// --- HELPER FUNCTION: Convert seconds (Real) to HHH:MM:SS string ---
FUNCTION "FC_SecondsToTimeString" : String[9]
{ S7_Optimized_Access := 'TRUE' }
VERSION : 0.1
	VAR_INPUT
		seconds : Real;
	END_VAR
	VAR_TEMP
		totalSec : DInt;
		hours : Int;
		minutes : Int;
		secs : Int;
		h1, h2, h3, m1, m2, s1, s2 : USInt;
	END_VAR
BEGIN
	// Convert to integer seconds
	totalSec := REAL_TO_DINT(seconds);

	// Calculate hours, minutes, seconds
	hours := DINT_TO_INT(totalSec / 3600);
	minutes := DINT_TO_INT((totalSec MOD 3600) / 60);
	secs := DINT_TO_INT(totalSec MOD 60);

	// Limit to 999:59:59 max display (over 41 days)
	IF hours > 999 THEN
		hours := 999;
		minutes := 59;
		secs := 59;
	END_IF;

	// Convert to ASCII digit values (digit type USInt, like in existing code)
	h1 := UINT_TO_USINT(hours / 100);
	h2 := UINT_TO_USINT((hours MOD 100) / 10);
	h3 := UINT_TO_USINT(hours MOD 10);
	m1 := UINT_TO_USINT(minutes / 10);
	m2 := UINT_TO_USINT(minutes MOD 10);
	s1 := UINT_TO_USINT(secs / 10);
	s2 := UINT_TO_USINT(secs MOD 10);

	// Build string "HHH:MM:SS" using BYTE_TO_CHAR like existing filename code
	#FC_SecondsToTimeString := CONCAT(IN1 := BYTE_TO_CHAR(48 + h1), IN2 := BYTE_TO_CHAR(48 + h2));
	#FC_SecondsToTimeString := CONCAT(IN1 := #FC_SecondsToTimeString, IN2 := BYTE_TO_CHAR(48 + h3));
	#FC_SecondsToTimeString := CONCAT(IN1 := #FC_SecondsToTimeString, IN2 := ':');
	#FC_SecondsToTimeString := CONCAT(IN1 := #FC_SecondsToTimeString, IN2 := BYTE_TO_CHAR(48 + m1));
	#FC_SecondsToTimeString := CONCAT(IN1 := #FC_SecondsToTimeString, IN2 := BYTE_TO_CHAR(48 + m2));
	#FC_SecondsToTimeString := CONCAT(IN1 := #FC_SecondsToTimeString, IN2 := ':');
	#FC_SecondsToTimeString := CONCAT(IN1 := #FC_SecondsToTimeString, IN2 := BYTE_TO_CHAR(48 + s1));
	#FC_SecondsToTimeString := CONCAT(IN1 := #FC_SecondsToTimeString, IN2 := BYTE_TO_CHAR(48 + s2));
END_FUNCTION

// --- LOGGING FUNCTION BLOCK ---
// Volani:
//   OB30 (1000ms): LogManager.SampleStep()   - plni buffer kazdych SampleEveryN_Cycles cyklu
//   Main (OB1):   LogManager.FlushPending   - zkontroluj flag a zapis na SD
FUNCTION_BLOCK "FB_LogManager"
{ S7_Optimized_Access := 'TRUE' }
VERSION : 0.1
	VAR_INPUT
		Enable : Bool;                     // povoleni logovani (z DB_LogConfig.Enable)
		StartTest : Bool;                  // hrana = start testu (z DB_LogConfig.StartTest)
		StopTest : Bool;                   // hrana = manual stop testu (z DB_LogConfig.StopTest)
		RPM : Real;                        // aktualni otacky vretene [RPM]
		T_Lozisko : Real;                  // teplota loziska [degC]
		T_Uhliky : Real;                   // teplota uhliku/kartacu [degC] – zatim 0.0
		Vibrace : Real;                    // vibrace – zatim 0.0
		ProudUhliky : Real;                // proud do uhliku [A], prepocitany z AQ1_CurrentCtrl_V
		State : USInt;                     // stav vretene: 0=STOP 1=RUN 2=STOPPING 3=TRIP
		RunLatched : Bool;                 // vreteno v provozu (latch z FB_DriveCtrl)
		TripActive : Bool;                 // safety trip aktivni
		TripCode : USInt;                  // kod tripu: 0=OK 1=ESTOP 2=RELAY 3=EXT 4=TEMP 5=VIB 6=DISABLE
		SafetyText : String[40];           // textova diagnostika safety brany
		SampleEveryN_Cycles : Int := 6;    // pocet cyklu OB30 mezi vzorky → 6×1s = 6s/vzorek
		TestDuration_s : DInt := 1814400;  // max delka testu [s] – timeout vypnut, beha do manualniko stopu
		FlushEveryN : Int := 5;            // pocet vzorku pred flushem: 5=test (30s), 100=produkce (10min)
		AckFlush : Bool;                   // potvrzeni flushe od FB_LogFlushToSd → resetuje FlushPending
	END_VAR

	VAR_OUTPUT
		FlushPending : Bool;       // TRUE = buffer ma dost dat → OB1 ma zapsat na SD
		TestTimeoutReached : Bool; // TRUE = test dosahl TestDuration_s (logika vypnuta)
		CyclesProcessed : DInt;    // pocet OB30 cyklu zpracovanych behem testu
		LastFlushTrigger : USInt;  // co spustilo posledni flush: 1=periodic 2=manual stop 3=timeout
		EdgeStopDetected : Bool;   // prave detekovan StopTest puls (jeden OB30 cyklus)
		EdgeStartDetected : Bool;  // prave detekovan StartTest puls (jeden OB30 cyklus)
	END_VAR

	VAR
		prevStartTest : Bool := FALSE;
		prevStopTest : Bool := FALSE;
		cycleCounter : Int := 0;
		flushCounter : Int := 0;
		StopReason : USInt := 0;  // 0=running, 1=manual stop, 2=timeout, 3=trip/fault
	END_VAR

	VAR_TEMP
		startDtl  : DTL;
		rdRet     : Int;
		yr2       : UInt;
		fName     : String[32];
		digit     : USInt;
	END_VAR

BEGIN
	// Detekce startu testu (hrana)
	EdgeStartDetected := FALSE;
	EdgeStopDetected := FALSE;

	IF Enable AND (StartTest AND NOT prevStartTest) THEN
		EdgeStartDetected := TRUE;  // Diagnostika
		"DB_LogRuntime".TestActive := TRUE;
		"DB_LogRuntime".StopSequenceActive := FALSE;
		"DB_LogRuntime".LastStopLogSaved := FALSE;
		"DB_LogRuntime".Elapsed_s := 0.0;
		"DB_LogRuntime".SampleCounter := 0;
		"DB_LogRuntime".FlushErrorCount := 0;
		"DB_LogRuntime".LastFlushOk := FALSE;  // Jeste neprobehl zadny flush
		"DB_LogRuntime".HeaderWritten := FALSE;
		"DB_LogBuffer".TrendWriteIdx := 0;
		"DB_LogBuffer".TrendReadIdx := 0;
		cycleCounter := 0;
		flushCounter := 0;
		FlushPending := FALSE;
		TestTimeoutReached := FALSE;
		CyclesProcessed := 0;  // Reset diagnostiky
		LastFlushTrigger := 0;

		// Format initial times for HMI display
		"DB_LogRuntime".ElapsedTime_HMI := '000:00:00';
		"DB_LogRuntime".TargetTime_HMI := "FC_SecondsToTimeString"(seconds := DINT_TO_REAL(TestDuration_s));

		// Generate timestamp-based file name using direct digit manipulation
		rdRet := RD_SYS_T(OUT := startDtl);

		// Build filename: LOG_YYMMDD_HHMMSS.csv
		fName := 'LOG_';

		// Year (last 2 digits)
		yr2 := startDtl.YEAR MOD 100;
		digit := UINT_TO_USINT(yr2 / 10);
		fName := CONCAT(IN1 := fName, IN2 := BYTE_TO_CHAR(48 + digit));
		digit := UINT_TO_USINT(yr2 MOD 10);
		fName := CONCAT(IN1 := fName, IN2 := BYTE_TO_CHAR(48 + digit));

		// Month
		digit := startDtl.MONTH / 10;
		fName := CONCAT(IN1 := fName, IN2 := BYTE_TO_CHAR(48 + digit));
		digit := startDtl.MONTH MOD 10;
		fName := CONCAT(IN1 := fName, IN2 := BYTE_TO_CHAR(48 + digit));

		// Day
		digit := startDtl.DAY / 10;
		fName := CONCAT(IN1 := fName, IN2 := BYTE_TO_CHAR(48 + digit));
		digit := startDtl.DAY MOD 10;
		fName := CONCAT(IN1 := fName, IN2 := BYTE_TO_CHAR(48 + digit));

		fName := CONCAT(IN1 := fName, IN2 := '_');

		// Hour
		digit := startDtl.HOUR / 10;
		fName := CONCAT(IN1 := fName, IN2 := BYTE_TO_CHAR(48 + digit));
		digit := startDtl.HOUR MOD 10;
		fName := CONCAT(IN1 := fName, IN2 := BYTE_TO_CHAR(48 + digit));

		// Minute
		digit := startDtl.MINUTE / 10;
		fName := CONCAT(IN1 := fName, IN2 := BYTE_TO_CHAR(48 + digit));
		digit := startDtl.MINUTE MOD 10;
		fName := CONCAT(IN1 := fName, IN2 := BYTE_TO_CHAR(48 + digit));

		// Second
		digit := startDtl.SECOND / 10;
		fName := CONCAT(IN1 := fName, IN2 := BYTE_TO_CHAR(48 + digit));
		digit := startDtl.SECOND MOD 10;
		fName := CONCAT(IN1 := fName, IN2 := BYTE_TO_CHAR(48 + digit));

		fName := CONCAT(IN1 := fName, IN2 := '.csv');

		"DB_LogRuntime".FileName := fName;
		"DB_LogRuntime".HeaderWritten := FALSE;
		"DB_LogRuntime".FlushErrorCount := 0;
		"DB_LogRuntime".LastFlushOk := FALSE;  // Jeste neprobehl zadny flush
		"DB_LogRuntime".MaxTempLozisko_C := 0.0;  // Reset max teploty pri startu testu
		"DB_LogRuntime".MaxTempUhliky_C := 0.0;   // Reset max teploty pri startu testu
		StopReason := 0;  // Reset stop reason - test běží
		// (event log: TEST_START)
	END_IF;

	// Detekce stopu testu (hrana)
	IF Enable AND (StopTest AND NOT prevStopTest) THEN
		EdgeStopDetected := TRUE;  // Diagnostika
		"DB_LogRuntime".StopSequenceActive := TRUE;
		"DB_LogRuntime".LastStopLogSaved := FALSE;
		StopReason := 1;  // Manual stop

		// Write final stop record before clearing TestActive so CSV captures stop state
		"DB_LogBuffer".TrendBuffer["DB_LogBuffer".TrendWriteIdx].t_s := "DB_LogRuntime".Elapsed_s;
		"DB_LogBuffer".TrendBuffer["DB_LogBuffer".TrendWriteIdx].RPM := RPM;
		"DB_LogBuffer".TrendBuffer["DB_LogBuffer".TrendWriteIdx].T_Lozisko := T_Lozisko;
		"DB_LogBuffer".TrendBuffer["DB_LogBuffer".TrendWriteIdx].T_Uhliky := T_Uhliky;
		"DB_LogBuffer".TrendBuffer["DB_LogBuffer".TrendWriteIdx].Vibrace := Vibrace;
		"DB_LogBuffer".TrendBuffer["DB_LogBuffer".TrendWriteIdx].ProudUhliky := ProudUhliky;
		"DB_LogBuffer".TrendBuffer["DB_LogBuffer".TrendWriteIdx].State := State;
		"DB_LogBuffer".TrendBuffer["DB_LogBuffer".TrendWriteIdx].RunLatched := RunLatched;
		"DB_LogBuffer".TrendBuffer["DB_LogBuffer".TrendWriteIdx].TripActive := TripActive;
		"DB_LogBuffer".TrendBuffer["DB_LogBuffer".TrendWriteIdx].TripCode := TripCode;
		"DB_LogBuffer".TrendBuffer["DB_LogBuffer".TrendWriteIdx].SafetyText := SafetyText;
		"DB_LogBuffer".TrendBuffer["DB_LogBuffer".TrendWriteIdx].TestActive := FALSE;
		"DB_LogBuffer".TrendBuffer["DB_LogBuffer".TrendWriteIdx].StopReason := StopReason;
		"DB_LogBuffer".TrendWriteIdx := "DB_LogBuffer".TrendWriteIdx + 1;
		IF "DB_LogBuffer".TrendWriteIdx > 999 THEN
			"DB_LogBuffer".TrendWriteIdx := 0;
		END_IF;

		"DB_LogRuntime".TestActive := FALSE;
		FlushPending := TRUE;   // finalni flush pri manuálním stopu
		LastFlushTrigger := 2;  // manual stop flush
		// (event log: TEST_STOP)
	END_IF;

	prevStartTest := StartTest;
	prevStopTest := StopTest;

	// Handshake: FB_LogFlushToSd potvrdil flush -> resetovat FlushPending
	// AckFlush zustane TRUE dokud FlushPending neklesne (4-way handshake)
	IF AckFlush THEN
		FlushPending := FALSE;
		flushCounter := 0;  // Reset counter az PO dokonceni flush-u
	END_IF;

	// Cyklické vzorkování pouze pokud test běží
	IF Enable AND "DB_LogRuntime".TestActive THEN
		cycleCounter := cycleCounter + 1;

		// Timer HMI se aktualizuje kazdy OB30 cyklus (1 s), nezavisle na vzorkovani logu.
		"DB_LogRuntime".Elapsed_s := "DB_LogRuntime".Elapsed_s + 1.0;
		"DB_LogRuntime".ElapsedTime_HMI := "FC_SecondsToTimeString"(seconds := "DB_LogRuntime".Elapsed_s);
		"DB_LogRuntime".TimeDisplay_HMI := CONCAT(
			IN1 := "DB_LogRuntime".ElapsedTime_HMI,
			IN2 := ' / '
		);
		"DB_LogRuntime".TimeDisplay_HMI := CONCAT(
			IN1 := "DB_LogRuntime".TimeDisplay_HMI,
			IN2 := "DB_LogRuntime".TargetTime_HMI
		);

		IF cycleCounter >= SampleEveryN_Cycles THEN
			cycleCounter := 0;

			// Zapis vzorku do kruhoveho bufferu
			"DB_LogBuffer".TrendBuffer["DB_LogBuffer".TrendWriteIdx].t_s := "DB_LogRuntime".Elapsed_s;
			"DB_LogBuffer".TrendBuffer["DB_LogBuffer".TrendWriteIdx].RPM := RPM;
			"DB_LogBuffer".TrendBuffer["DB_LogBuffer".TrendWriteIdx].T_Lozisko := T_Lozisko;
			"DB_LogBuffer".TrendBuffer["DB_LogBuffer".TrendWriteIdx].T_Uhliky := T_Uhliky;
			"DB_LogBuffer".TrendBuffer["DB_LogBuffer".TrendWriteIdx].Vibrace := Vibrace;
			"DB_LogBuffer".TrendBuffer["DB_LogBuffer".TrendWriteIdx].ProudUhliky := ProudUhliky;
			"DB_LogBuffer".TrendBuffer["DB_LogBuffer".TrendWriteIdx].State := State;
			"DB_LogBuffer".TrendBuffer["DB_LogBuffer".TrendWriteIdx].RunLatched := RunLatched;
			"DB_LogBuffer".TrendBuffer["DB_LogBuffer".TrendWriteIdx].TripActive := TripActive;
			"DB_LogBuffer".TrendBuffer["DB_LogBuffer".TrendWriteIdx].TripCode := TripCode;
			"DB_LogBuffer".TrendBuffer["DB_LogBuffer".TrendWriteIdx].SafetyText := SafetyText;
			"DB_LogBuffer".TrendBuffer["DB_LogBuffer".TrendWriteIdx].TestActive := "DB_LogRuntime".TestActive;
			"DB_LogBuffer".TrendBuffer["DB_LogBuffer".TrendWriteIdx].StopReason := StopReason;

			// Update maximalni teploty behem testu
			IF T_Lozisko > "DB_LogRuntime".MaxTempLozisko_C THEN
				"DB_LogRuntime".MaxTempLozisko_C := T_Lozisko;
			END_IF;
			IF T_Uhliky > "DB_LogRuntime".MaxTempUhliky_C THEN
				"DB_LogRuntime".MaxTempUhliky_C := T_Uhliky;
			END_IF;

			// Posun indexu (kruhový buffer)
			"DB_LogBuffer".TrendWriteIdx := "DB_LogBuffer".TrendWriteIdx + 1;
			IF "DB_LogBuffer".TrendWriteIdx > 999 THEN
				"DB_LogBuffer".TrendWriteIdx := 0;
			END_IF;
			"DB_LogRuntime".SampleCounter := "DB_LogRuntime".SampleCounter + 1;

			// FlushPending: Main vi, ze je cas zapsat na SD
			flushCounter := flushCounter + 1;
			IF flushCounter >= FlushEveryN AND NOT FlushPending THEN
				FlushPending := TRUE;
				LastFlushTrigger := 1;  // periodic flush
			END_IF;
		END_IF;

		// Konec testu po uplynutí času - VYPNUTO (test bezi do nekonecna, az do manualniho stopu)
		// IF "DB_LogRuntime".Elapsed_s >= DINT_TO_REAL(TestDuration_s) THEN
		// 	"DB_LogRuntime".TestActive := FALSE;
		// 	StopReason := 2;  // Timeout
		// 	TestTimeoutReached := TRUE;
		// 	FlushPending := TRUE;   // posledni flush
		// 	LastFlushTrigger := 3;  // timeout flush
		// 	// (event log: TEST_END_TIMEOUT)
		// END_IF;

		CyclesProcessed := CyclesProcessed + 1;  // Diagnostika
	END_IF;
END_FUNCTION_BLOCK
TYPE "UDT_SENSORS"
VERSION : 0.1
   STRUCT
      AI1_Teplota_Lozisko_C : Real;
      AI2_Teplota_Kartace_C : Real;
      TM_Rotation_A_Channel : Real;
   END_STRUCT;


END_TYPE

// --- LOGGING UDTs ---
TYPE "UDT_LogRecord"
VERSION : 0.1
	STRUCT
		t_s : Real;
		RPM : Real;
		T_Lozisko : Real;
		T_Uhliky : Real;
		Vibrace : Real;
		ProudUhliky : Real;
		State : USInt;
		RunLatched : Bool;
		TripActive : Bool;
		TripCode : USInt;
		SafetyText : String[40];
		TestActive : Bool;    // TRUE = test běží, FALSE = test byl zastaven
		StopReason : USInt;   // 0=běží, 1=manual stop, 2=timeout, 3=trip/fault
	END_STRUCT;
END_TYPE

TYPE "UDT_EventRecord"
VERSION : 0.1
	STRUCT
		t_s : Real;
		EventCode : USInt;
		EventText : String[32];
		State : USInt;
		TripCode : USInt;
		SafetyText : String[40];
	END_STRUCT;
END_TYPE

FUNCTION "FC_LogRecordToCsv" : String[254]
{ S7_Optimized_Access := 'TRUE' }
VERSION : 0.1
	VAR_INPUT
		Rec : "UDT_LogRecord";
	END_VAR

	VAR_TEMP
		line : String[254];
	END_VAR

BEGIN
	line := REAL_TO_STRING(Rec.t_s);
	line := CONCAT(IN1 := line, IN2 := ',');
	line := CONCAT(IN1 := line, IN2 := REAL_TO_STRING(Rec.RPM));
	line := CONCAT(IN1 := line, IN2 := ',');
	line := CONCAT(IN1 := line, IN2 := REAL_TO_STRING(Rec.T_Lozisko));
	line := CONCAT(IN1 := line, IN2 := ',');
	line := CONCAT(IN1 := line, IN2 := REAL_TO_STRING(Rec.T_Uhliky));
	line := CONCAT(IN1 := line, IN2 := ',');
	line := CONCAT(IN1 := line, IN2 := REAL_TO_STRING(Rec.Vibrace));
	line := CONCAT(IN1 := line, IN2 := ',');
	line := CONCAT(IN1 := line, IN2 := REAL_TO_STRING(Rec.ProudUhliky));
	line := CONCAT(IN1 := line, IN2 := ',');
	line := CONCAT(IN1 := line, IN2 := USINT_TO_STRING(Rec.State));
	line := CONCAT(IN1 := line, IN2 := ',');

	IF Rec.RunLatched THEN
		line := CONCAT(IN1 := line, IN2 := '1');
	ELSE
		line := CONCAT(IN1 := line, IN2 := '0');
	END_IF;

	line := CONCAT(IN1 := line, IN2 := ',');
	IF Rec.TripActive THEN
		line := CONCAT(IN1 := line, IN2 := '1');
	ELSE
		line := CONCAT(IN1 := line, IN2 := '0');
	END_IF;

	line := CONCAT(IN1 := line, IN2 := ',');
	line := CONCAT(IN1 := line, IN2 := USINT_TO_STRING(Rec.TripCode));
	line := CONCAT(IN1 := line, IN2 := ',');
	line := CONCAT(IN1 := line, IN2 := Rec.SafetyText);
	line := CONCAT(IN1 := line, IN2 := ',');

	IF Rec.TestActive THEN
		line := CONCAT(IN1 := line, IN2 := '1');
	ELSE
		line := CONCAT(IN1 := line, IN2 := '0');
	END_IF;

	line := CONCAT(IN1 := line, IN2 := ',');
	line := CONCAT(IN1 := line, IN2 := USINT_TO_STRING(Rec.StopReason));

	#FC_LogRecordToCsv := #line;
END_FUNCTION

DATA_BLOCK "DB_LogConfig"
{ S7_Optimized_Access := 'TRUE' }
VERSION : 0.1
NON_RETAIN
	VAR
		Enable : Bool;             // TRUE = logovani povoleno (default TRUE)
		StartTest : Bool;          // HMI/WebAPI: nastav TRUE pro start testu (hrana, auto-reset OB30)
		StopTest : Bool;           // HMI/WebAPI: nastav TRUE pro manual stop testu (hrana, auto-reset OB30)
		TestDuration_s : DInt;     // max delka testu [s] – default 1814400 = 3 tydny
		FlushEveryN : Int;         // flush kazdych N vzorku – default 5 (30s), prod 100 (10min)
		FilePrefix : String[16];   // rezerva pro pojmenovani souboru (zatim nevyuzito)
	END_VAR
BEGIN
	Enable := TRUE;
	StartTest := false;
	StopTest := false;
	TestDuration_s := 1814400;  // 3 tydny = 21 dni = 504 hodin
	FlushEveryN := 5;  // TESTOVACI NASTAVENI (prod: 100)
	FilePrefix := 'testlog';
END_DATA_BLOCK

DATA_BLOCK "DB_LogRuntime"
{ S7_Optimized_Access := 'TRUE' }
VERSION : 0.2
NON_RETAIN
	VAR
		TestActive : Bool;             // TRUE = test probiha (sleduj pro zahajeni mereni)
		TestActivePrev : Bool;         // predchozi stav TestActive pro edge logiku v OB1
		StartReqLatched : Bool;        // OB1 latch StartTest pulsu (ochrana proti ztrate hrany pri OB30=1000ms)
		StopReqLatched : Bool;         // OB1 latch StopTest pulsu (ochrana proti ztrate hrany pri OB30=1000ms)
		StopSequenceActive : Bool;     // TRUE = probiha stop sekvence a ceka se na final flush
		LastStopLogSaved : Bool;       // TRUE = posledni stop dokoncil flush na SD (indikace pro HMI)
		TestStartTs : Date_And_Time;   // cas startu testu (RD_SYS_T pri StartTest hrane)
		Elapsed_s : Real;              // uplynuly cas od startu testu [s], aktualizuje se kazdou 1s
		SampleCounter : DInt;          // celkovy pocet vzorku zapsanych do bufferu od startu
		LastFlushOk : Bool;            // TRUE = posledni flush na SD probehl bez chyby
		LastError : String[40];        // text posledni chyby flushe (FileWriteC status kod)
		FileName : String[32];         // nazev aktualniho log souboru (LOG_YYMMDD_HHMMSS.csv)
		HeaderWritten : Bool;          // TRUE = CSV hlavicka uz zapsana do souboru
		FlushErrorCount : Int;         // pocet chyb flushe od posledniho startu (alarm >0)
		// HMI display strings (formatted time)
		ElapsedTime_HMI : String[9];   // HMI zobrazeni uplynuteho casu "HHH:MM:SS" (max 999h)
		TargetTime_HMI : String[9];    // HMI zobrazeni ciloveho casu "HHH:MM:SS"
		TimeDisplay_HMI : String[21];  // HMI jedno pole: "HHH:MM:SS / HHH:MM:SS"
		// Maximalni teploty behem testu
		MaxTempLozisko_C : Real;       // max teplota loziska od startu testu [degC]
		MaxTempUhliky_C : Real;        // max teplota uhliku/kartacu od startu testu [degC]
		// OB30 cycle time monitoring
		OB30_LastTs : DTL;             // posledni cas zacatku OB30 cyklu
		OB30_CycleTime_ms : Int;       // delka aktualniho OB30 cyklu [ms]
		OB30_MaxCycleTime_ms : Int;    // maximum vzorkovany cyklus [ms]
		OB30_MinCycleTime_ms : Int;    // minimum vzorkovany cyklus [ms] (init 1000)
		OB30_AverageCycleTime_ms : Real; // prumer platnych OB30 cyklu [ms]
		OB30_CycleTimeOutOfRange : Bool; // TRUE = prumer mimo 950..1050 ms pro HMI
		OB30_CycleTimeSum_ms : Real;   // pomocny soucet platnych OB30 mereni [ms]
		OB30_CycleCounter : DInt;      // pocet OB30 cyklu od startu testu (kazdych 1s by se zvysil o 1)
	END_VAR
BEGIN
	TestActive := false;
	TestActivePrev := false;
	StartReqLatched := false;
	StopReqLatched := false;
	StopSequenceActive := false;
	LastStopLogSaved := false;
	Elapsed_s := 0.0;
	SampleCounter := 0;
	LastFlushOk := false;  // Jeste neprobehl zadny flush
	LastError := '';
	FileName := '';
	HeaderWritten := false;
	FlushErrorCount := 0;
	ElapsedTime_HMI := '000:00:00';
	TargetTime_HMI := '000:00:00';
	TimeDisplay_HMI := '000:00:00 / 000:00:00';
	MaxTempLozisko_C := 0.0;
	MaxTempUhliky_C := 0.0;
	OB30_CycleTime_ms := 0;
	OB30_MaxCycleTime_ms := 0;
	OB30_MinCycleTime_ms := 1000;
	OB30_AverageCycleTime_ms := 0.0;
	OB30_CycleTimeOutOfRange := FALSE;
	OB30_CycleTimeSum_ms := 0.0;
	OB30_CycleCounter := 0;
END_DATA_BLOCK

DATA_BLOCK "DB_LogBuffer"
{ S7_Optimized_Access := 'TRUE' }
VERSION : 0.1
NON_RETAIN
	VAR
		TrendBuffer : ARRAY[0..999] OF "UDT_LogRecord";   // kruhovy buffer vzorku (1000 polozek × 6s = 100 min)
		EventBuffer : ARRAY[0..99] OF "UDT_EventRecord";  // buffer eventu (faze 3)
		TrendWriteIdx : Int;   // index zapisu (LogManager) – sleduj pro debug plneni bufferu
		TrendReadIdx : Int;    // index cteni/flushe (LogFlushToSd) – WriteIdx-ReadIdx = neprectenych radku
		EventWriteIdx : Int;   // index zapisu eventu
		EventReadIdx : Int;    // index cteni eventu
	END_VAR
BEGIN
	TrendWriteIdx := 0;
	TrendReadIdx := 0;
	EventWriteIdx := 0;
	EventReadIdx := 0;
END_DATA_BLOCK

DATA_BLOCK "DB_HMI"
{ S7_Optimized_Access := 'TRUE' }
VERSION : 0.1
NON_RETAIN
   VAR
      Sensors { S7_SetPoint := 'False'} : "UDT_SENSORS";   // AI hodnoty po prepoctu (teploty degC, RPM)
      System : Struct
         Enable : Bool;   // rezerva pro systemove povoleni
      END_STRUCT;
      Spindle : Struct
         Start : Bool;    // HMI puls start vretene (auto-reset v OB1)
         Stop : Bool;     // HMI puls stop vretene (auto-reset v OB1)
         ResetFault : Bool;  // HMI puls reset chyby meniče
         Speed_RPM : Real;   // zadane otacky vretene [RPM] – max 18000
         Enable : Bool;      // rezerva
      END_STRUCT;
      LabPSU : Struct
         Enable : Bool;            // povoleni laboratorniho zdroje (auto-set pri StartTest)
			Cycle_s : Real;           // perioda OB30 [s] – default 1.0
			Mode : USInt;             // rezim zdroje: 0=OFF 1=CONST 2=SINE_DEBUG
			BaseVoltage_V : Real;     // napeti zdroje [V] – default 2.0
			DebugAmplitude_A : Real;  // amplituda sinusoidy [A] – default 5.0
			DebugPeriod_min : Real;   // perioda sinusoidy [min] – default 1.0 min
			CurrentOffset_A : Real;   // deprecated: v SINE_DEBUG se nepouziva
			ConstCurrent_A : Real;    // proud v CONST rezimu [A] – default 10.0
			MaxCurrent_A : Real;      // maximalni povoleny proud [A] – default 38.0
			CurrentLimitExceeded : Bool;  // TRUE = zadany proud prekrocil MaxCurrent_A
			SineCycleCounter : UDInt;     // pocet dokoncenych period sinusoidy od startu
      END_STRUCT;
   END_VAR


BEGIN
	LabPSU.Enable := false;
	LabPSU.Cycle_s := 1.0;  // OB30 = 1000ms = 1s
	LabPSU.Mode := 2;  // 2 = SINE_DEBUG (sinusova modulace)
	LabPSU.BaseVoltage_V := 2.0;
	LabPSU.DebugAmplitude_A := 5.0;
	LabPSU.DebugPeriod_min := 1.0;  // 1 minuta perioda
	LabPSU.CurrentOffset_A := 5.0;
	LabPSU.ConstCurrent_A := 10.0;  // 10 A pro CONST rezim
	LabPSU.MaxCurrent_A := 38.0;
	LabPSU.CurrentLimitExceeded := false;
	LabPSU.SineCycleCounter := 0;

END_DATA_BLOCK

TYPE "UDT_TM_COUNT"
VERSION : 0.1
   STRUCT
      MeasuredValue : Real;
   END_STRUCT;

END_TYPE

TYPE "UDT_IO_AQ"
VERSION : 0.1
   STRUCT
      SpeedVoltage : Real;
      AQ2_VoltageCtrl_V : Real;
      AQ1_CurrentCtrl_V : Real;
		AQ3_OutputOff : Real;
   END_STRUCT;

END_TYPE

TYPE "UDT_IO_AI"
VERSION : 0.1
   STRUCT
      AI1_TeplotaLoziska_Ohm : Int;
      AI2_TeplotaKartace_Ohm : Int;
   END_STRUCT;

END_TYPE

TYPE "UDT_IO_DI"
VERSION : 0.1
   STRUCT
      SafetyRelayAuxOk : Bool;
      HSC_Couter : UInt;
      EmergencyStop : Bool;
      ExternalFault : Bool;
   END_STRUCT;

END_TYPE

TYPE "UDT_IO_DQ"
VERSION : 0.1
   STRUCT
      EmergencyStop : Bool;
      EmergencyStopButtonLed : Bool;
      ResetButtonLed : Bool;
      RunForwardCmd : Bool;
      FaultResetCmd : Bool;
      MultiSpeed1 : Bool;
      ExternalFault : Bool;
   END_STRUCT;

END_TYPE

FUNCTION_BLOCK "FB_SafetyGate"
{ S7_Optimized_Access := 'TRUE' }
VERSION : 0.1
   VAR_INPUT
      Enable : Bool;   // hlavní povolení systému
      EmergencyStop : Bool;   // 1 = E-Stop aktivní
      SafetyRelayAuxOk : Bool;   // 1 = safety relé OK
      ExternalFault : Bool;   // 1 = externí chyba
      TempAlarm : Bool;   // 1 = kritická teplota
      VibAlarm : Bool;   // 1 = kritické vibrace
   END_VAR

   VAR_OUTPUT
      SafetyOk : Bool;
      PermitMotion : Bool;
      TripActive : Bool;
      TripCode : USInt;
      StatusText : String[40];
   END_VAR


BEGIN
	// hardware safety stav
	#SafetyOk := #SafetyRelayAuxOk AND NOT #EmergencyStop;

	// centrální trip
	#TripActive := (NOT #SafetyOk) OR #ExternalFault OR #TempAlarm OR #VibAlarm OR (NOT #Enable);

	// povolení pohybu
	#PermitMotion := NOT #TripActive;

	// diagnostika
	IF #EmergencyStop THEN
	    #TripCode := 1;
	    #StatusText := 'E-STOP ACTIVE';
	ELSE
		IF NOT #SafetyRelayAuxOk THEN
		    #TripCode := 2;
		    #StatusText := 'SAFETY RELAY NOT OK';
		ELSE
			IF #ExternalFault THEN
			    #TripCode := 3;
			    #StatusText := 'EXTERNAL FAULT';
			ELSE
				IF #TempAlarm THEN
				    #TripCode := 4;
				    #StatusText := 'TEMP ALARM';
				ELSE
					IF #VibAlarm THEN
					    #TripCode := 5;
					    #StatusText := 'VIBRATION ALARM';
					ELSE
						IF NOT #Enable THEN
						    #TripCode := 6;
						    #StatusText := 'SYSTEM NOT ENABLED';
						ELSE
						    #TripCode := 0;
						    #StatusText := 'READY';
						END_IF;
					END_IF;
				END_IF;
			END_IF;
		END_IF;
	END_IF;
END_FUNCTION_BLOCK

FUNCTION_BLOCK "FB_LabPSU"
{ S7_Optimized_Access := 'TRUE' }
VERSION : 0.1
   VAR_INPUT
      Enable : Bool := false;   // povolenÃ­ funkce z PLC/HMI
      PermitOutput : Bool := false;   // interlock / safety gate
      Mode : USInt := 0;   // 0=OFF, 1=CONST, 2=SINE_DEBUG ÄasovÃ¡ zÃ¡kladna
      Cycle_s : Real := 0.01;   // typicky OB35 = 10 ms zdroj - zÃ¡kladnÃ­ nastavenÃ­
      BaseVoltage_V : Real := 1.0;   // AQ2
      CurrentOffset_A : Real := 0.0;   // DC offset proudu
      DebugAmplitude_A : Real := 60.0;   // amplituda sinu pro debug
      DebugPeriod_min : Real := 10.0;   // perioda sinu v minutach (default 10 min)
      ConstCurrent_A : Real := 10.0;   // rampy
      RampUp_A_per_s : Real := 50.0;
      RampDown_A_per_s : Real := 80.0;   // parametry zdroje BK1900B
	PSU_MinVoltage_V : Real := 0.8;   // minimalni napeti pro stabilni vystup zdroje
      PSU_MaxVoltage_V : Real := 16.0;   // model 1900B
      PSU_MaxCurrent_A : Real := 60.0;   // model 1900B
      RemoteMaxCtrl_V : Real := 5.0;   // analog remote 0..5 V engineering outputs
   END_VAR

   VAR_OUTPUT
      VoltageSet_V : Real := 0.0;   // poÅ¾adovanÃ© napÄ›tÃ­ zdroje
      CurrentSet_A : Real := 0.0;   // poÅ¾adovanÃ½ current limit analog outputs for PLC IO layer
      AQ2_VoltageCtrl_V : Real := 0.0;   // 0..5 V na pin 2
      AQ3_CurrentCtrl_V : Real := 0.0;   // 0..5 V na pin 3 digital output for pin 5
	AQ_OutputOff_V : Real := 5.0;   // 0.0 V = enable, 5.0 V = output off
      State : USInt := 0;   // 0 OFF, 1 CONST, 2 SINE
      StatusText : String[40] := '';
      CurrentLimitExceeded : Bool := false;   // indikator, ze uzivatel zkusil zadat vyssi proud nez limit
      SineCycleCounter : UDInt := 0;   // pocet dokoncenych period sinusovky (pro HMI)
   END_VAR

   VAR
      phase_rad : Real := 0.0;
      omega : Real := 0.0;
      targetCurrent_A : Real := 0.0;
      sineValue : Real := 0.0;
	effectiveOffset_A : Real := 0.0;
	offsetAutoAdjusted : Bool := FALSE;
	prevMode : USInt := 0;   // Pamatuje si predchozi Mode pro detekci prechodu
   END_VAR


BEGIN
	// safety / permit
	IF (NOT #Enable) OR (NOT #PermitOutput) THEN
	    #phase_rad := 0.0;
	    #VoltageSet_V := 0.0;
	    #CurrentSet_A := 0.0;
	    #AQ2_VoltageCtrl_V := 0.0;
	    #AQ3_CurrentCtrl_V := 0.0;
	    #AQ_OutputOff_V := 5.0;
	    #State := 0;
	    #StatusText := 'SAFE OFF';
	    #CurrentLimitExceeded := false;
	    #prevMode := 0;
	    RETURN;
	END_IF;

	// reset CurrentLimitExceeded flag na zacatku cyklu
	#CurrentLimitExceeded := false;

	// vystup zdroje povolen
	#AQ_OutputOff_V := 0.0;

	// zakladni napeti
	#VoltageSet_V := #BaseVoltage_V;

	// omezeni napeti
	IF #VoltageSet_V < #PSU_MinVoltage_V THEN
	    #VoltageSet_V := #PSU_MinVoltage_V;
	END_IF;
	IF #VoltageSet_V > #PSU_MaxVoltage_V THEN
	    #VoltageSet_V := #PSU_MaxVoltage_V;
	END_IF;

	CASE #Mode OF
	    0: // OFF
	        #CurrentSet_A := 0.0;
	        #VoltageSet_V := 0.0;
	        #AQ_OutputOff_V := 5.0;
	        #State := 0;
	        #StatusText := 'OFF';

	    1: // CONST
	        #targetCurrent_A := #ConstCurrent_A;

	        // detekce prekroceni limitu - pred clampingem
	        IF #targetCurrent_A > #PSU_MaxCurrent_A THEN
	            #CurrentLimitExceeded := true;
	        END_IF;

	        IF #targetCurrent_A < 0.0 THEN
	            #targetCurrent_A := 0.0;
	        END_IF;
	        IF #targetCurrent_A > #PSU_MaxCurrent_A THEN
	            #targetCurrent_A := #PSU_MaxCurrent_A;
	        END_IF;

	        // jednoducha rampa
	        IF #CurrentSet_A < #targetCurrent_A THEN
	            #CurrentSet_A := #CurrentSet_A + (#RampUp_A_per_s * #Cycle_s);
	            IF #CurrentSet_A > #targetCurrent_A THEN
	                #CurrentSet_A := #targetCurrent_A;
	            END_IF;
	        ELSE
			IF #CurrentSet_A > #targetCurrent_A THEN
			    #CurrentSet_A := #CurrentSet_A - (#RampDown_A_per_s * #Cycle_s);
			    IF #CurrentSet_A < #targetCurrent_A THEN
			        #CurrentSet_A := #targetCurrent_A;
			    END_IF;
			END_IF;
	        END_IF;

	        #State := 1;
	        #StatusText := 'CONST';

	    2: // SINE_DEBUG
	        // Pri prvnim vstupu do SINE rezimu resetovat fazi na -pi/2, aby prubeh zacinali od 0A
	        IF #prevMode <> 2 THEN
	            #phase_rad := -1.5707963;  // -pi/2 rad, zacatek prubehu od 0 A
	            #SineCycleCounter := 0;  // reset pocitadla cyklu pri vstupu do SINE rezimu
	        END_IF;

	        // Vypocet omega z periody v minutach: omega = 2*pi / (T_min * 60)
	        IF #DebugPeriod_min > 0.0 THEN
	            #omega := 6.2831853 / (#DebugPeriod_min * 60.0); // 2*pi / (T_min * 60s)
	        ELSE
	            #omega := 0.0; // ochrana proti deleni nulou
	        END_IF;
	        #offsetAutoAdjusted := FALSE;
	        IF #prevMode <> 2 THEN
	            // Prvni vypocet po vstupu do rezimu zacne presne na 0 A.
	            #phase_rad := -1.5707963 - (#omega * #Cycle_s);
	        END_IF;

	        #phase_rad := #phase_rad + (#omega * #Cycle_s);

	        // drzet fazi v rozumnem rozsahu a pocitat dokoncene periody
	        IF #phase_rad > 6.2831853 THEN
	            #phase_rad := #phase_rad - 6.2831853;
	            #SineCycleCounter := #SineCycleCounter + 1;  // dokoncena jedna perioda
	        END_IF;

	        #sineValue := SIN(#phase_rad);

	        // Cely sinus posunuty do rozsahu 0..A.
	        // DebugAmplitude_A je maximum prubehu, CurrentOffset_A se v SINE_DEBUG nepouziva.
	        #targetCurrent_A := (#DebugAmplitude_A * 0.5)
	                          + ((#DebugAmplitude_A * 0.5) * #sineValue);

	        // detekce prekroceni limitu - pred clampingem
	        IF #targetCurrent_A > #PSU_MaxCurrent_A THEN
	            #CurrentLimitExceeded := true;
	        END_IF;

	        // current limit zdroje nemuze byt zaporny
	        IF #targetCurrent_A < 0.0 THEN
	            #targetCurrent_A := 0.0;
	        END_IF;

	        IF #targetCurrent_A > #PSU_MaxCurrent_A THEN
	            #targetCurrent_A := #PSU_MaxCurrent_A;
	        END_IF;

	        // volitelne muzes i tady nechat rampu, ale pro sinus ji vetsinou nechces moc agresivni
	        #CurrentSet_A := #targetCurrent_A;

	        #State := 2;
	        #StatusText := 'SINE DEBUG 0..A';

	    ELSE
	        #CurrentSet_A := 0.0;
	        #VoltageSet_V := 0.0;
	        #AQ_OutputOff_V := 5.0;
	        #State := 0;
	        #StatusText := 'UNKNOWN->OFF';
	END_CASE;

	// prevod engineering units -> BK remote control 0..5V

	// napeti
	IF #PSU_MaxVoltage_V > 0.0 THEN
	    #AQ2_VoltageCtrl_V := (#VoltageSet_V / #PSU_MaxVoltage_V) * #RemoteMaxCtrl_V;
	ELSE
	    #AQ2_VoltageCtrl_V := 0.0;
	END_IF;

	// proud - kalibrovany prepocet na zaklade mereni
	// I [A] = 15.92 * U [V] - 6.09  ->  U [V] = (I [A] / 15.92) + 0.383
	// Dead zone: 0.383 V
	IF #CurrentSet_A > 0.0 THEN
	    #AQ3_CurrentCtrl_V := (#CurrentSet_A / 15.92) + 0.383;
	ELSE
	    #AQ3_CurrentCtrl_V := 0.0;
	END_IF;

	// clamp
	IF #AQ2_VoltageCtrl_V < 0.0 THEN
	    #AQ2_VoltageCtrl_V := 0.0;
	END_IF;
	IF #AQ2_VoltageCtrl_V > #RemoteMaxCtrl_V THEN
	    #AQ2_VoltageCtrl_V := #RemoteMaxCtrl_V;
	END_IF;

	// clamp proudoveho ridiciho signalu
	// Dead zone: pod 0.383V zdroj nereaguje
	IF #AQ3_CurrentCtrl_V < 0.0 THEN
	    #AQ3_CurrentCtrl_V := 0.0;
	END_IF;
	IF #AQ3_CurrentCtrl_V > #RemoteMaxCtrl_V THEN
	    #AQ3_CurrentCtrl_V := #RemoteMaxCtrl_V;
	END_IF;

	// Ulozit aktualni Mode pro detekci prechodu v pristim cyklu
	#prevMode := #Mode;

END_FUNCTION_BLOCK

TYPE "UDT_LABPSU_STATUS"
VERSION : 0.1
   STRUCT
      VoltageSet_V : Real;
      CurrentSet_A : Real;
      State : USInt;
      StatusText : String[40];
   END_STRUCT;

END_TYPE

TYPE "UDT_SAFETY_STATUS"
VERSION : 0.1
   STRUCT
      SafetyOk : Bool;
      PermitMotion : Bool;
      TripActive : Bool;
      TripCode : USInt;
      StatusText : String[40];
   END_STRUCT;

END_TYPE

DATA_BLOCK "DB_IO"
{ S7_Optimized_Access := 'TRUE' }
VERSION : 0.1
NON_RETAIN
   VAR
      DQ { S7_SetPoint := 'False'} : "UDT_IO_DQ";
      DI : "UDT_IO_DI";
      AI : "UDT_IO_AI";
      TM : "UDT_TM_COUNT";
      AQ : "UDT_IO_AQ";
   END_VAR


BEGIN
	AQ.AQ3_OutputOff := 5.0;

END_DATA_BLOCK

TYPE "UDT_SPINDEL_STATUS"
VERSION : 0.1
   STRUCT
      RunLatched : Bool;
      TripActive : Bool;
      State : USInt;
      StatusText : String[40];
   END_STRUCT;

END_TYPE

FUNCTION_BLOCK "FB_DriveCtrl"
{ S7_Optimized_Access := 'TRUE' }
VERSION : 0.1
   VAR_INPUT
      HMI_Start : Bool := false;   // start command (button)
      HMI_Stop : Bool := false;   // stop command (button)
      HMI_ResetFault : Bool := false;   // reset fault (button)
      HMI_Speed_RPM : Real := 0.0;   // speed setpoint in RPM Interlocks / safety
      PermitMotion : Bool := false;   // from safety gate
      EmergencyStop : Bool := false;   // E-Stop chain
      ExternalFaultIn : Bool := false;   // external fault input Parameters
      SpeedMax_RPM : Real := 18000.0;   // max RPM corresponds to 10V
      AO_MaxVolt : Real := 10.0;   // 0..10V
      RampUp_RPM_per_s : Real := 6000.0;   // ramp up rate
      RampDown_RPM_per_s : Real := 9000.0;   // ramp down rate
      ResetPulse : Time := T#300MS;   // reset pulse length
      RequireSpeedToRun : Bool := FALSE;   // if TRUE, Start only latches when setpoint > 0 Outputs to drive
   END_VAR

   VAR_OUTPUT
      DO_RunForward : Bool := false;
      DO_FaultReset : Bool := false;
      DO_MultiSpeed1 : Bool := false;
      DO_ExternalFault : Bool := false;
      AQ1_Voltage_0_10V : Real := 0.0;   // Status for HMI/diagnostics
      RunLatched : Bool := false;   // internal run request latch
      TripActive : Bool := false;   // interlock active
      State : USInt := 0;   // 0 STOPPED, 1 RUN_CMD, 2 STOPPING, 3 TRIP
      StatusText : String[40] := '';   // Edge detection
   END_VAR

   VAR
      prevStart : Bool := false;
      prevStop : Bool := false;
      prevReset : Bool := false;
      startEdge : Bool := false;
      stopEdge : Bool := false;
      resetEdge : Bool := false;   // Ramp variables
      speedCmdRPM : Real := 0.0;
      speedRampRPM : Real := 0.0;   // Reset pulse timer
      tReset {InstructionName := 'TON_TIME'; LibVersion := '1.0'; S7_SetPoint := 'False'} : TON_TIME;   // Cycle time assumption (OB1). Use OB35 for precise timing if needed.
      cycle_s { S7_SetPoint := 'True'} : Real := 0.01;   // 10 ms default
   END_VAR


BEGIN
	    // ------------------------------------------------------------
	    // Edge detection for Start/Stop/Reset
	    // ------------------------------------------------------------
	    #startEdge := #HMI_Start AND NOT #prevStart;
	    #stopEdge := #HMI_Stop AND NOT #prevStop;
	    #resetEdge := #HMI_ResetFault AND NOT #prevReset;

	    #prevStart := #HMI_Start;
	    #prevStop := #HMI_Stop;
	    #prevReset := #HMI_ResetFault;

	    // ------------------------------------------------------------
	    // Trip / interlock
	    // Trip znamena zakaz běhu vřetene, pokud není splněna bezpečnostní podmínka. Trip = okamžité odstavení zařízení.
	    // ------------------------------------------------------------
	    #TripActive := (NOT #PermitMotion) OR #EmergencyStop OR #ExternalFaultIn;

	    // External fault output to the drive (if wired this way)
	    #DO_ExternalFault := #TripActive;

	    // ------------------------------------------------------------
	    // Sanitize setpoint
	    // Sanitize = zkontrolovat a upravit vstupní hodnotu tak, aby byla bezpečná a platná.
	    // ------------------------------------------------------------
	    #speedCmdRPM := #HMI_Speed_RPM;
	    IF #speedCmdRPM < 0.0 THEN
	        #speedCmdRPM := 0.0;
	    END_IF;
	    IF #speedCmdRPM > #SpeedMax_RPM THEN
	        #speedCmdRPM := #SpeedMax_RPM;
	    END_IF;

	    // ------------------------------------------------------------
	    // Run latch logic (Stop has priority)
	    // ------------------------------------------------------------
	    IF #TripActive THEN
	        #RunLatched := FALSE;
	    ELSE
	        IF #stopEdge OR #HMI_Stop THEN
	            #RunLatched := FALSE;
	        ELSE
	            IF #startEdge THEN
	                IF (NOT #RequireSpeedToRun) OR (#speedCmdRPM > 0.0) THEN
	                    #RunLatched := TRUE;
	                END_IF;
	            END_IF;
	        END_IF;
	    END_IF;

	    // ------------------------------------------------------------
	    // Fault reset pulse (recommended only when not running)
	    // ------------------------------------------------------------
	    #tReset(IN := (#resetEdge AND NOT #TripActive AND NOT #RunLatched),
	            PT := #ResetPulse);
	    #DO_FaultReset := #tReset.Q;

	    // ------------------------------------------------------------
	    // Defaults
	    // ------------------------------------------------------------
	    #DO_MultiSpeed1 := FALSE;

	    // ------------------------------------------------------------
	    // State (for HMI readability; no drive feedback available)
	    // ------------------------------------------------------------
	    IF #TripActive THEN
	        #State := 3; // TRIP
	    ELSE
	        IF #RunLatched THEN
	            #State := 1; // RUN_CMD
	        ELSE
	            IF #speedRampRPM > 0.0 THEN
	                #State := 2; // STOPPING (ramp down)
	            ELSE
	                #State := 0; // STOPPED
	            END_IF;
	        END_IF;
	    END_IF;

	    CASE #State OF
	        0:
	            #StatusText := 'STOPPED';
	        1:
	            #StatusText := 'RUN CMD (no feedback)';
	        2:
	            #StatusText := 'STOPPING (ramp down)';
	        3:
	            #StatusText := 'TRIP (E-Stop/Interlock)';
	        ELSE
	            #StatusText := 'UNKNOWN';
	    END_CASE;

	    // ------------------------------------------------------------
	    // Drive command + speed ramp
	    // ------------------------------------------------------------
	    IF #TripActive THEN
	        #DO_RunForward := FALSE;
	        #speedRampRPM := 0.0;
	    ELSE
	        IF #RunLatched THEN
	            #DO_RunForward := TRUE;

	            // Ramp toward setpoint (up & down)
	            IF #speedRampRPM < #speedCmdRPM THEN
	                #speedRampRPM := #speedRampRPM + (#RampUp_RPM_per_s * #cycle_s);
	                IF #speedRampRPM > #speedCmdRPM THEN
	                    #speedRampRPM := #speedCmdRPM;
	                END_IF;
	            ELSE
				IF #speedRampRPM > #speedCmdRPM THEN
				    #speedRampRPM := #speedRampRPM - (#RampDown_RPM_per_s * #cycle_s);
				    IF #speedRampRPM < #speedCmdRPM THEN
				        #speedRampRPM := #speedCmdRPM;
				    END_IF;
				END_IF;
	            END_IF;

	        ELSE
	            #DO_RunForward := FALSE;

	            // Ramp down to 0
	            IF #speedRampRPM > 0.0 THEN
	                #speedRampRPM := #speedRampRPM - (#RampDown_RPM_per_s * #cycle_s);
	                IF #speedRampRPM < 0.0 THEN
	                    #speedRampRPM := 0.0;
	                END_IF;
	            END_IF;
	        END_IF;
	    END_IF;

	    // ------------------------------------------------------------
	    // RPM -> 0..10V conversion
	    // ------------------------------------------------------------
	    IF #SpeedMax_RPM > 0.0 THEN
	        #AQ1_Voltage_0_10V := (#speedRampRPM / #SpeedMax_RPM) * #AO_MaxVolt;
	    ELSE
	        #AQ1_Voltage_0_10V := 0.0;
	    END_IF;

	    // ------------------------------------------------------------
	    // Clamp AO (Clamp znamena omezit hodnotu tak, aby zůstala v daném rozsahu (min–max))
	    //  ------------------------------------------------------------
	    IF #AQ1_Voltage_0_10V < 0.0 THEN
	        #AQ1_Voltage_0_10V := 0.0;
	    END_IF;
	    IF #AQ1_Voltage_0_10V > #AO_MaxVolt THEN
	        #AQ1_Voltage_0_10V := #AO_MaxVolt;
	    END_IF;

	    // Hard safety
	    IF #TripActive THEN
	        #AQ1_Voltage_0_10V := 0.0;
	    END_IF;

END_FUNCTION_BLOCK

FUNCTION_BLOCK "FB_SafetyButtons"
{ S7_Optimized_Access := 'TRUE' }
VERSION : 0.1
   VAR_INPUT
      DI0_AuxSafetyRelay : Bool;   // AUX ze safety relé
      DI1_SafetyButton : Bool;   // signal ze safety tlačítka
   END_VAR

   VAR_OUTPUT
      DQ1_LED : Bool;   // Cervene LED svetlo na STOP tlacitku
      DQ0_LED : Bool;   // Modre LED reset svetlo
   END_VAR


BEGIN
	// Bezpečný default
	#DQ1_LED := FALSE;
	#DQ0_LED := FALSE;

	// Vyhodnocení kombinací
	IF (NOT #DI0_AuxSafetyRelay) AND (#DI1_SafetyButton) THEN
	    // DI0 = 0, DI1 = 0
	    #DQ1_LED := TRUE;
	    #DQ0_LED := FALSE;

	ELSE
		IF (NOT #DI0_AuxSafetyRelay) AND (NOT #DI1_SafetyButton) THEN
		    // DI0 = 0, DI1 = 1
		    #DQ1_LED := FALSE;
		    #DQ0_LED := TRUE;

		ELSE
			IF #DI0_AuxSafetyRelay AND (NOT #DI1_SafetyButton) THEN
			    // DI0 = 1, DI1 = 1
			    #DQ1_LED := FALSE;
			    #DQ0_LED := FALSE;

			ELSE
				// DI0 = 1, DI1_SafetyButton = true -> relay OK, button stisknuty = E-STOP fault stav
				// cervena LED sviti
				#DQ1_LED := TRUE;
				#DQ0_LED := FALSE;
			END_IF;
		END_IF;
	END_IF;
END_FUNCTION_BLOCK

DATA_BLOCK "DB_Status"
{ S7_Optimized_Access := 'TRUE' }
VERSION : 0.1
NON_RETAIN
   VAR
      Spindel { S7_SetPoint := 'False'} : "UDT_SPINDEL_STATUS";
      Safety : "UDT_SAFETY_STATUS";
      LabPSU { S7_SetPoint := 'False'} : "UDT_LABPSU_STATUS";
      // HMI helper for status panel color (Basic Panel limitation - one tag only)
	HMI_StatusColor : USInt;  // 0=READY (green), 1=RUNNING (blue), 2=RED (error/trip), 3=AMBER (running with RPM=0)
	HMI_StatusText : String[24];  // "TEST READY" / "TEST RUNNING" / "RUNNING - RPM=0" / "READY - LOG SAVED" / "ERROR - TRIP ACTIVE"
   END_VAR


BEGIN
   HMI_StatusColor := 0;
   HMI_StatusText := 'TEST READY';
END_DATA_BLOCK

DATA_BLOCK "FB_SafetyButtons_DB"
{ S7_Optimized_Access := 'TRUE' }
VERSION : 0.1
NON_RETAIN
"FB_SafetyButtons"

BEGIN

END_DATA_BLOCK

DATA_BLOCK "Spindel"
{ S7_Optimized_Access := 'TRUE' }
VERSION : 0.1
NON_RETAIN
"FB_DriveCtrl"

BEGIN

END_DATA_BLOCK

DATA_BLOCK "TM_Counter"
{InstructionName := 'High_Speed_Counter';
 LibVersion := '5.0';
 S7_Optimized_Access := 'TRUE' }
AUTHOR : SIMATIC
FAMILY : HSC
NAME : HSC
VERSION : 5.0
NON_RETAIN
High_Speed_Counter

BEGIN
   Configuration.HWID := 263;
   Configuration.ChannelNo := 0;
   Configuration.CounterInputs.SignalType := 0;
   Configuration.CounterInputs.FilterFrequency := 3;

END_DATA_BLOCK

DATA_BLOCK "LabPSU"
{ S7_Optimized_Access := 'TRUE' }
VERSION : 0.1
NON_RETAIN
"FB_LabPSU"

BEGIN

END_DATA_BLOCK

DATA_BLOCK "Safety_1"
{ S7_Optimized_Access := 'TRUE' }
VERSION : 0.1
NON_RETAIN
"FB_SafetyGate"

BEGIN

END_DATA_BLOCK

DATA_BLOCK "DB_Alarms"
{ S7_Optimized_Access := 'TRUE' }
VERSION : 0.1
NON_RETAIN
   VAR
	TempHighLozisko : Bool;   // TRUE = teplota loziska > TempHighLoziskoThreshold_C
	TempHighKartace : Bool;   // TRUE = teplota kartacu > TempHighKartaceThreshold_C
      TempAlarm : Bool;         // TRUE = TempHighLozisko OR TempHighKartace → trip
      VibCritical : Bool;       // TRUE = kritické vibrace (senzor zatim nezapojen)
   END_VAR


BEGIN

END_DATA_BLOCK

DATA_BLOCK "DB_Config"
{ S7_Optimized_Access := 'TRUE' }
VERSION : 0.1
NON_RETAIN
	VAR
		TempHighThreshold_C : Real;   // deprecated: legacy common threshold
		TempHighLoziskoThreshold_C : Real;   // prah teploty loziska [degC]
		TempHighKartaceThreshold_C : Real;   // prah teploty kartace [degC]
		VibCriticalThreshold : Real;  // prahova hodnota vibraci – default 0.0 (senzor nezapojen)
		DAC_MaxDacRange : Int;        // max hodnota DAC pro 10V (S7-1200) – default 27648
		InputSim : Struct
			EnableSafetyRelayAuxOverride : Bool;   // SIM: TRUE = pouzij SafetyRelayAuxOk misto fyzickeho DI0
			SafetyRelayAuxOk : Bool;               // SIM default TRUE – simuluje OK safety rele (PermitMotion=TRUE)
			EnableEmergencyStopOverride : Bool;    // SIM: TRUE = pouzij EmergencyStop misto fyzickeho DI1
			EmergencyStop : Bool;                  // SIM default FALSE – simuluje uvolneny E-Stop (bez tripu)
			EnableRPM_Sim : Bool;                  // SIM: TRUE = pouzij SimRPM misto TM_Counter
			SimRPM : Real;                         // SIM default 12000.0 RPM (max 18000)
			EnableTempLozisko_Sim : Bool;          // SIM: TRUE = pouzij SimTempLozisko_C misto AI1_RTD
			SimTempLozisko_C : Real;               // SIM default 35.0 degC (alarm >65 degC)
			EnableTempKartace_Sim : Bool;          // SIM: TRUE = pouzij SimTempKartace_C misto AI2_RTD
			SimTempKartace_C : Real;               // SIM default 40.0 degC (alarm >65 degC)
		END_STRUCT;
	END_VAR

BEGIN
	TempHighThreshold_C := 65.0;
	TempHighLoziskoThreshold_C := 65.0;
	TempHighKartaceThreshold_C := 65.0;
	VibCriticalThreshold := 0.0;
	DAC_MaxDacRange := 27648;
	InputSim.EnableSafetyRelayAuxOverride := false;
	InputSim.SafetyRelayAuxOk := true;
	InputSim.EnableEmergencyStopOverride := false;
	InputSim.EmergencyStop := false;
	InputSim.EnableRPM_Sim := false;
	InputSim.SimRPM := 12000.0;
	InputSim.EnableTempLozisko_Sim := false;
	InputSim.SimTempLozisko_C := 35.0;
	InputSim.EnableTempKartace_Sim := false;
	InputSim.SimTempKartace_C := 40.0;

END_DATA_BLOCK

FUNCTION "FC_ConvertIO" : Void
{ S7_Optimized_Access := 'TRUE' }
VERSION : 0.1

BEGIN
	IF "DB_Config".InputSim.EnableTempLozisko_Sim THEN
		"DB_HMI".Sensors.AI1_Teplota_Lozisko_C := "DB_Config".InputSim.SimTempLozisko_C;
	ELSE
		"DB_HMI".Sensors.AI1_Teplota_Lozisko_C := "DB_IO".AI.AI1_TeplotaLoziska_Ohm / 10.0;
	END_IF;
	IF "DB_Config".InputSim.EnableTempKartace_Sim THEN
		"DB_HMI".Sensors.AI2_Teplota_Kartace_C := "DB_Config".InputSim.SimTempKartace_C;
	ELSE
		"DB_HMI".Sensors.AI2_Teplota_Kartace_C := "DB_IO".AI.AI2_TeplotaKartace_Ohm / 10.0;
	END_IF;
	IF "DB_Config".InputSim.EnableRPM_Sim THEN
		"DB_HMI".Sensors.TM_Rotation_A_Channel := "DB_Config".InputSim.SimRPM;
	ELSE
		"DB_HMI".Sensors.TM_Rotation_A_Channel := ("DB_IO".TM.MeasuredValue * 60) / 2;
	END_IF;
END_FUNCTION

FUNCTION "FC_IO_Map_Write" : Void
{ S7_Optimized_Access := 'TRUE' }
VERSION : 0.1

BEGIN
	"AQ0" := REAL_TO_INT("DB_IO".AQ.SpeedVoltage / 10.0 * 27648.0);
	"AQ1" := REAL_TO_INT("DB_IO".AQ.AQ1_CurrentCtrl_V / 10.0 * 27648.0);
	"AQ2" := REAL_TO_INT("DB_IO".AQ.AQ2_VoltageCtrl_V / 10.0 * 27648.0);
	"AQ3" := REAL_TO_INT("DB_IO".AQ.AQ3_OutputOff / 10.0 * 27648.0);

	"DQ0_MI1_Run_Forward" := "DB_IO".DQ.RunForwardCmd;
	"DQ1_Reset_Button_Blue_LED" := "DB_IO".DQ.ResetButtonLed;
	"DQ2_Stop_Button_Red_Led" := "DB_IO".DQ.EmergencyStopButtonLed;
END_FUNCTION

FUNCTION "FC_IO_Map_Read" : Void
{ S7_Optimized_Access := 'TRUE' }
VERSION : 0.1

BEGIN
	IF "DB_Config".InputSim.EnableSafetyRelayAuxOverride THEN
		"DB_IO".DI.SafetyRelayAuxOk := "DB_Config".InputSim.SafetyRelayAuxOk;
	ELSE
		"DB_IO".DI.SafetyRelayAuxOk := "DI0_SafetyRelay_Aux";
	END_IF;
	IF "DB_Config".InputSim.EnableEmergencyStopOverride THEN
		"DB_IO".DI.EmergencyStop := "DB_Config".InputSim.EmergencyStop;
	ELSE
		"DB_IO".DI.EmergencyStop := NOT "DI1_SafetyRelay_Released_Safety_Button"; // DI1_SafetyRelay_Released_Safety_Button = False znamena, ze mame stisknuty safety button, ktery je normally closed a po stisknuti se kontakt rozpoji a na vstupu je 0V
	END_IF;
	"DB_IO".AI.AI1_TeplotaLoziska_Ohm := "AI1_RTD";
	"DB_IO".AI.AI2_TeplotaKartace_Ohm := "AI2_RTD";
END_FUNCTION

DATA_BLOCK "FB_LabPSU_DB"
{ S7_Optimized_Access := 'TRUE' }
VERSION : 0.1
NON_RETAIN
"FB_LabPSU"

BEGIN

END_DATA_BLOCK

DATA_BLOCK "LogManager"
{ S7_Optimized_Access := 'TRUE' }
VERSION : 0.1
NON_RETAIN
"FB_LogManager"

BEGIN

END_DATA_BLOCK

FUNCTION_BLOCK "FB_LogFlushToSd"
{ S7_Optimized_Access := 'TRUE' }
VERSION : 0.1
	VAR_INPUT
		Enable : Bool;                    // povoleni flushe (z DB_LogConfig.Enable)
		FlushRequest : Bool;              // pozadavek na flush (z LogManager.FlushPending)
		FinalFlush : Bool;                // TRUE = zapsat vse bez limitu (pri manual stopu)
		MaxRowsPerFlush : Int := 50;      // max radku na jeden flush (50 = ~5s pri 10 FileWriteC/s)
		RetryLimit : Int := 3;            // max pokusu po chybe pred nastavenim Error=TRUE
	END_VAR

	VAR_OUTPUT
		Busy : Bool;               // TRUE = flush probiha (stavovy automat mimo IDLE)
		AckFlush : Bool;           // potvrzeni flushe pro LogManager (drzi TRUE dokud FlushRequest neklesne)
		Error : Bool;              // TRUE = flush selhal po vsech retry pokusech
		ErrorCode : Word;          // posledni FileWriteC status kod (napr. 0x7001=soubor neexistuje)
		CurrentStep : USInt;       // aktualni krok automatu: 0=IDLE 1=PREP 2=OPEN 3=HDR 4=ROW 5=NEXT 6=CLOSE 7=ACK 10=ERR 11=MKDIR
		RowsFlushed : Int;         // pocet radku zapsanych pri poslednim flushu
	END_VAR

	VAR
		Step : USInt;
		RowIdx : Int;
		RowsToFlush : Int;
		RowsDone : Int;
		RetryCount : Int;
		prevFlushReq : Bool;
		writeReq : Bool;
		writeStarted : Bool;
		filePath : String[64];
		CsvLine : String[254];
		CsvBytes : Array[0..253] of Byte;
		writeOffset : UDInt;
		fileOffset_Bytes : UDInt;
		writeLength : UDInt;
		writeResultLength : UDInt;
		fwDone : Bool;
		fwBusy : Bool;
		fwError : Bool;
		dirCreated : Bool := FALSE;  // Flag pro sledovani, zda byla slozka vytvorena
		dirCreateStarted : Bool;

		FileWriteC_1 {InstructionName := 'FileWriteC'; LibVersion := '1.0'} : FileWriteC;
		FileWriteC_DirKeeper {InstructionName := 'FileWriteC'; LibVersion := '1.0'} : FileWriteC;  // Pro vytvoreni slozky
		FileStatus : Word;
	END_VAR

	VAR_TEMP
		rowsAvail : Int;
		csvLen : Int;
		i : Int;
	END_VAR

	VAR CONSTANT
		STEP_IDLE : USInt := 0;
		STEP_PREPARE : USInt := 1;
		STEP_CREATE_DIR : USInt := 11;  // Novy stav pro vytvoreni slozky
		STEP_OPEN : USInt := 2;
		STEP_WR_HEADER : USInt := 3;
		STEP_WR_ROW : USInt := 4;
		STEP_NEXT_ROW : USInt := 5;
		STEP_CLOSE : USInt := 6;
		STEP_ACK : USInt := 7;
		STEP_ERROR : USInt := 10;
	END_VAR

BEGIN
	// AckFlush is NOT reset here – STEP_IDLE holds it until FlushRequest drops (4-way handshake)
	CurrentStep := Step;  // Diagnostika - exportovat aktualni krok

	CASE Step OF
		STEP_IDLE:
			Busy := FALSE;
			Error := FALSE;
			writeReq := FALSE;
			writeStarted := FALSE;
			// Hold AckFlush TRUE until FlushRequest drops so OB30 (1000ms) can see it
			IF NOT FlushRequest THEN
				AckFlush := FALSE;
			END_IF;
			IF Enable AND (FlushRequest AND NOT prevFlushReq) THEN
				Busy := TRUE;
				Step := STEP_PREPARE;
			END_IF;

		STEP_PREPARE:
			IF "DB_LogBuffer".TrendWriteIdx >= "DB_LogBuffer".TrendReadIdx THEN
				rowsAvail := "DB_LogBuffer".TrendWriteIdx - "DB_LogBuffer".TrendReadIdx;
			ELSE
				rowsAvail := (1000 - "DB_LogBuffer".TrendReadIdx) + "DB_LogBuffer".TrendWriteIdx;
			END_IF;

			IF FinalFlush THEN
				RowsToFlush := rowsAvail;
			ELSE
				RowsToFlush := rowsAvail;
				IF RowsToFlush > MaxRowsPerFlush THEN
					RowsToFlush := MaxRowsPerFlush;
				END_IF;
			END_IF;

			IF RowsToFlush <= 0 THEN
				Step := STEP_ACK;
			ELSE
				RowIdx := "DB_LogBuffer".TrendReadIdx;
				RowsDone := 0;
				RetryCount := 0;
				filePath := CONCAT(IN1 := 'UserFiles/', IN2 := "DB_LogRuntime".FileName);
				// Pokud slozka jeste nebyla vytvorena, zkus ji vytvorit nejdriv
				IF NOT dirCreated THEN
					Step := STEP_CREATE_DIR;
				ELSE
					Step := STEP_OPEN;
				END_IF;
			END_IF;

		STEP_CREATE_DIR:
			// Vytvoreni slozky UserFiles pomoci zapisu prazdneho keep souboru
			IF NOT dirCreateStarted THEN
				CsvBytes[0] := 0;  // Prazdny obsah
				writeReq := TRUE;
				dirCreateStarted := TRUE;
			END_IF;

			FileWriteC_DirKeeper(
				REQ := writeReq,
				Name := 'UserFiles/.keepdir',  // Pomocny soubor pro vytvoreni slozky
				Offset := 0,
				Length := 1,
				Done => fwDone,
				Busy => fwBusy,
				Error => fwError,
				Status => FileStatus,
				ResultLength => writeResultLength,
				Data := CsvBytes
			);

			writeReq := FALSE;

			IF fwDone THEN
				// Slozka uspesne vytvorena (nebo uz existovala)
				dirCreated := TRUE;
				dirCreateStarted := FALSE;
				writeStarted := FALSE;
				Step := STEP_OPEN;
			ELSIF fwError THEN
				// Chyba pri vytvareni - pokracuj dale, mozna slozka uz existuje
				// Nebo to zkus bez slozky
				IF FileStatus = 16#7002 OR FileStatus = 16#0000 OR FileStatus = 16#7000 THEN
					// 0x7002 = uz existuje, 0x7000 = generic warning - to je OK
					dirCreated := TRUE;
				END_IF;
				dirCreateStarted := FALSE;
				writeStarted := FALSE;
				Step := STEP_OPEN;
			ELSIF NOT fwBusy AND dirCreateStarted THEN
				// FileWriteC skoncil (Busy=FALSE) ale nenastavil Done ani Error
				// Tento stav muze nastat pri 16#7000 (warning misto error)
				// Pokracuj dale, pravdepodobne slozka existuje
				dirCreated := TRUE;
				dirCreateStarted := FALSE;
				writeStarted := FALSE;
				Step := STEP_OPEN;
			END_IF;

		STEP_OPEN:
			IF LEN(filePath) = 0 THEN
				FileStatus := 16#8001;
				Step := STEP_ERROR;
			ELSE
				IF NOT "DB_LogRuntime".HeaderWritten THEN
					fileOffset_Bytes := 0;
				END_IF;
				IF "DB_LogRuntime".HeaderWritten THEN
					Step := STEP_WR_ROW;
				ELSE
					Step := STEP_WR_HEADER;
				END_IF;
			END_IF;

		STEP_WR_HEADER:
			IF NOT writeStarted THEN
				CsvLine := 't_s,RPM,T_Lozisko,T_Uhliky,Vibrace,ProudUhliky,State,RunLatched,TripActive,TripCode,SafetyText,TestActive,StopReason';
				csvLen := LEN(CsvLine);
				FOR i := 0 TO 253 DO
					CsvBytes[i] := 0;
				END_FOR;
				FOR i := 1 TO csvLen DO
					CsvBytes[i - 1] := CHAR_TO_BYTE(CsvLine[i]);
				END_FOR;
				// Add CRLF (0x0D, 0x0A) for line ending
				CsvBytes[csvLen] := 13;
				CsvBytes[csvLen + 1] := 10;
				writeOffset := fileOffset_Bytes;
				writeLength := INT_TO_UDINT(csvLen + 2);
				writeReq := TRUE;
				writeStarted := TRUE;
			END_IF;

			FileWriteC_1(
				REQ := writeReq,
				Name := filePath,
				Offset := writeOffset,
				Length := writeLength,
				Done => fwDone,
				Busy => fwBusy,
				Error => fwError,
				Status => FileStatus,
				ResultLength => writeResultLength,
				Data := CsvBytes
			);

			writeReq := FALSE;

			IF fwDone THEN
				fileOffset_Bytes := fileOffset_Bytes + writeResultLength;
				"DB_LogRuntime".HeaderWritten := TRUE;
				writeStarted := FALSE;
				Step := STEP_WR_ROW;
			ELSE
				IF fwError THEN
					writeStarted := FALSE;
					Step := STEP_ERROR;
				END_IF;
			END_IF;

		STEP_WR_ROW:
			IF NOT writeStarted THEN
				CsvLine := "FC_LogRecordToCsv"(Rec := "DB_LogBuffer".TrendBuffer[RowIdx]);
				csvLen := LEN(CsvLine);
				FOR i := 0 TO 253 DO
					CsvBytes[i] := 0;
				END_FOR;
				FOR i := 1 TO csvLen DO
					CsvBytes[i - 1] := CHAR_TO_BYTE(CsvLine[i]);
				END_FOR;
				// Add CRLF (0x0D, 0x0A) for line ending
				CsvBytes[csvLen] := 13;
				CsvBytes[csvLen + 1] := 10;
				writeOffset := fileOffset_Bytes;
				writeLength := INT_TO_UDINT(csvLen + 2);
				writeReq := TRUE;
				writeStarted := TRUE;
			END_IF;

			FileWriteC_1(
				REQ := writeReq,
				Name := filePath,
				Offset := writeOffset,
				Length := writeLength,
				Done => fwDone,
				Busy => fwBusy,
				Error => fwError,
				Status => FileStatus,
				ResultLength => writeResultLength,
				Data := CsvBytes
			);

			writeReq := FALSE;

			IF fwDone THEN
				fileOffset_Bytes := fileOffset_Bytes + writeResultLength;
				writeStarted := FALSE;
				Step := STEP_NEXT_ROW;
			ELSE
				IF fwError THEN
					writeStarted := FALSE;
					Step := STEP_ERROR;
				END_IF;
			END_IF;

		STEP_NEXT_ROW:
			RowsDone := RowsDone + 1;
			RowIdx := RowIdx + 1;
			IF RowIdx >= 1000 THEN
				RowIdx := 0;
			END_IF;

			IF RowsDone >= RowsToFlush THEN
				Step := STEP_CLOSE;
			ELSE
				Step := STEP_WR_ROW;
			END_IF;

		STEP_CLOSE:
			Step := STEP_ACK;

		STEP_ACK:
			"DB_LogBuffer".TrendReadIdx := "DB_LogBuffer".TrendReadIdx + RowsDone;
			IF "DB_LogBuffer".TrendReadIdx >= 1000 THEN
				"DB_LogBuffer".TrendReadIdx := "DB_LogBuffer".TrendReadIdx - 1000;
			END_IF;
			"DB_LogRuntime".LastFlushOk := TRUE;
			RowsFlushed := RowsDone;  // Diagnostika
			AckFlush := TRUE;
			Busy := FALSE;
			Error := FALSE;
			Step := STEP_IDLE;

		STEP_ERROR:
			"DB_LogRuntime".LastFlushOk := FALSE;
			"DB_LogRuntime".FlushErrorCount := "DB_LogRuntime".FlushErrorCount + 1;
			"DB_LogRuntime".LastError := CONCAT(IN1 := 'FILEWRITEC STATUS ', IN2 := UINT_TO_STRING(WORD_TO_UINT(FileStatus)));
			ErrorCode := FileStatus;

			// Pokud je chyba 0x7001 (soubor/slozka neexistuje) a jeste jsme nezkusili vytvorit slozku
			IF (FileStatus = 16#7001) AND NOT dirCreated THEN
				// Zkus vytvorit slozku a pak retry
				writeStarted := FALSE;
				Step := STEP_CREATE_DIR;
			ELSE
				// Standardni retry logika
				RetryCount := RetryCount + 1;
				IF RetryCount <= RetryLimit THEN
					Step := STEP_OPEN;
				ELSE
					Error := TRUE;
					Busy := FALSE;
					AckFlush := TRUE;
					Step := STEP_IDLE;
				END_IF;
			END_IF;
	END_CASE;

	prevFlushReq := FlushRequest;
END_FUNCTION_BLOCK

DATA_BLOCK "LogFlushToSd"
{ S7_Optimized_Access := 'TRUE' }
VERSION : 0.1
NON_RETAIN
"FB_LogFlushToSd"

BEGIN

END_DATA_BLOCK

ORGANIZATION_BLOCK OB30
TITLE = "Cyclic Interrupt - 1000ms"
{ S7_Optimized_Access := 'TRUE' }
VERSION : 0.1
	VAR_TEMP
		currentTs : DTL;
		secNow_ms : DInt;
		secLast_ms : DInt;
		deltaMs : DInt;
		retVal : Int;
	END_VAR

BEGIN
	// Measure OB30 cycle time using RD_SYS_T()
	retVal := RD_SYS_T(currentTs);
	IF retVal = 0 AND "DB_LogRuntime".OB30_LastTs.NANOSECOND > 0 THEN
		// Cast USInt SECOND to DInt before multiply, then subtract to avoid type range error
		secNow_ms  := USINT_TO_DINT(currentTs.SECOND) * 1000 + UDINT_TO_DINT(currentTs.NANOSECOND / 1000000);
		secLast_ms := USINT_TO_DINT("DB_LogRuntime".OB30_LastTs.SECOND) * 1000 + UDINT_TO_DINT("DB_LogRuntime".OB30_LastTs.NANOSECOND / 1000000);
		deltaMs := secNow_ms - secLast_ms;
		IF deltaMs < 0 THEN deltaMs := deltaMs + 60000; END_IF;  // minute rollover (59→0)
		IF deltaMs > 32767 THEN deltaMs := 32767; END_IF;
		"DB_LogRuntime".OB30_CycleTime_ms := DINT_TO_INT(deltaMs);
		"DB_LogRuntime".OB30_CycleTimeSum_ms := "DB_LogRuntime".OB30_CycleTimeSum_ms
			+ INT_TO_REAL("DB_LogRuntime".OB30_CycleTime_ms);
		"DB_LogRuntime".OB30_CycleCounter := "DB_LogRuntime".OB30_CycleCounter + 1;
		"DB_LogRuntime".OB30_AverageCycleTime_ms :=
			"DB_LogRuntime".OB30_CycleTimeSum_ms
			/ DINT_TO_REAL("DB_LogRuntime".OB30_CycleCounter);
		"DB_LogRuntime".OB30_CycleTimeOutOfRange :=
			("DB_LogRuntime".OB30_AverageCycleTime_ms < 950.0)
			OR ("DB_LogRuntime".OB30_AverageCycleTime_ms > 1050.0);
		IF "DB_LogRuntime".OB30_CycleTime_ms > "DB_LogRuntime".OB30_MaxCycleTime_ms THEN
			"DB_LogRuntime".OB30_MaxCycleTime_ms := "DB_LogRuntime".OB30_CycleTime_ms;
		END_IF;
		IF "DB_LogRuntime".OB30_CycleTime_ms < "DB_LogRuntime".OB30_MinCycleTime_ms THEN
			"DB_LogRuntime".OB30_MinCycleTime_ms := "DB_LogRuntime".OB30_CycleTime_ms;
		END_IF;
	END_IF;
	IF retVal = 0 THEN
		"DB_LogRuntime".OB30_LastTs := currentTs;
	END_IF;

	// LabPSU - Current control (1s cycle time)
	"LabPSU"(Enable := "DB_HMI".LabPSU.Enable AND "DB_LogRuntime".TestActive,
	         PermitOutput := "DB_Status".Safety.PermitMotion,
	         Mode := "DB_HMI".LabPSU.Mode,
	         Cycle_s := 1.0,  // 1s cycle time (OB30 = 1000ms)
	         BaseVoltage_V := "DB_HMI".LabPSU.BaseVoltage_V,
	         CurrentOffset_A := "DB_HMI".LabPSU.CurrentOffset_A,
	         DebugAmplitude_A := "DB_HMI".LabPSU.DebugAmplitude_A,
	         DebugPeriod_min := "DB_HMI".LabPSU.DebugPeriod_min,
	         ConstCurrent_A := "DB_HMI".LabPSU.ConstCurrent_A,
	         RampUp_A_per_s := 50.0,
	         RampDown_A_per_s := 80.0,
	         PSU_MinVoltage_V := 0.8,
	         PSU_MaxVoltage_V := 16.0,
	         PSU_MaxCurrent_A := "DB_HMI".LabPSU.MaxCurrent_A,
	         RemoteMaxCtrl_V := 5.0,
	         VoltageSet_V => "DB_Status".LabPSU.VoltageSet_V,
	         CurrentSet_A => "DB_Status".LabPSU.CurrentSet_A,
	         AQ2_VoltageCtrl_V => "DB_IO".AQ.AQ2_VoltageCtrl_V,
	         AQ3_CurrentCtrl_V => "DB_IO".AQ.AQ1_CurrentCtrl_V,
	         AQ_OutputOff_V => "DB_IO".AQ.AQ3_OutputOff,
	         State => "DB_Status".LabPSU.State,
	         StatusText => "DB_Status".LabPSU.StatusText,
	         CurrentLimitExceeded => "DB_HMI".LabPSU.CurrentLimitExceeded,
	         SineCycleCounter => "DB_HMI".LabPSU.SineCycleCounter);

	// Logovani - vzorkovani kazdou 1s, SampleEveryN=6 -> 6s vzorek
	// File I/O (FlushPending) se zpracovava v Main (OB1), ne zde
	"LogManager"(
		Enable := "DB_LogConfig".Enable,
		StartTest := "DB_LogConfig".StartTest OR "DB_LogRuntime".StartReqLatched,
		StopTest := "DB_LogConfig".StopTest OR "DB_LogRuntime".StopReqLatched,
		RPM := "DB_HMI".Sensors.TM_Rotation_A_Channel,
		T_Lozisko := "DB_HMI".Sensors.AI1_Teplota_Lozisko_C,
		T_Uhliky := "DB_HMI".Sensors.AI2_Teplota_Kartace_C,
		Vibrace := 0.0,       // TODO: napojit na skutecny senzor vibraci
		ProudUhliky := "DB_Status".LabPSU.CurrentSet_A,
		State := "DB_Status".Spindel.State,
		RunLatched := "DB_Status".Spindel.RunLatched,
		TripActive := "DB_Status".Safety.TripActive,
		TripCode := "DB_Status".Safety.TripCode,
		SafetyText := "DB_Status".Safety.StatusText,
		SampleEveryN_Cycles := 6,
		TestDuration_s := "DB_LogConfig".TestDuration_s,
		FlushEveryN := "DB_LogConfig".FlushEveryN,
		AckFlush := "LogFlushToSd".AckFlush
	);

	//******************************************************************
	// AUTO-RESET pulse bits (provádí se každou 1s, AŽ PO LogManager)
	// Aby LogManager stihl detekovat hranu před resetem!
	//******************************************************************
	IF "LogManager".EdgeStartDetected THEN
		"DB_LogConfig".StartTest := FALSE;
		"DB_LogRuntime".StartReqLatched := FALSE;
	END_IF;
	IF "LogManager".EdgeStopDetected THEN
		"DB_LogConfig".StopTest := FALSE;
		"DB_LogRuntime".StopReqLatched := FALSE;
	END_IF;
END_ORGANIZATION_BLOCK

ORGANIZATION_BLOCK OB1
TITLE = "Main Program Sweep (Cycle)"
{ S7_Optimized_Access := 'TRUE' }
VERSION : 0.1
   VAR_TEMP
      WwwRetVal : Int;
   END_VAR


BEGIN
	//******************************************************************
	// IO MAP READ
	//******************************************************************
	"FC_IO_Map_Read"();
	"TM_Counter"(SwGate:=TRUE,
	             CaptureEnable:=FALSE,
	             SyncEnable:=FALSE,
	             ErrorAck:=FALSE,
	             EventAck:=FALSE,
	             MeasuredValue => "DB_IO".TM.MeasuredValue);

	// POZOR: FC_ConvertIO se volá AŽ na konci OB1, po všech FB!

	//******************************************************************
	// CALL FB BLOCKS - PRODUCTION LOGIC
	//******************************************************************
	"DB_Alarms".TempHighLozisko := "DB_HMI".Sensors.AI1_Teplota_Lozisko_C > "DB_Config".TempHighLoziskoThreshold_C;
	"DB_Alarms".TempHighKartace := "DB_HMI".Sensors.AI2_Teplota_Kartace_C > "DB_Config".TempHighKartaceThreshold_C;
	"DB_Alarms".TempAlarm := "DB_Alarms".TempHighLozisko OR "DB_Alarms".TempHighKartace;

	// Nektere safety signaly nemame implementovane - teplota, vibrace. Zatim bude potreba je simulovat
	"Safety_1"(Enable:= TRUE, // This signal can be used to bind to another system in the future
	           EmergencyStop:="DB_IO".DI.EmergencyStop,
	           SafetyRelayAuxOk:= "DB_IO".DI.SafetyRelayAuxOk,
	           ExternalFault:= "DB_IO".DI.ExternalFault,
	           TempAlarm:="DB_Alarms".TempAlarm,
	           VibAlarm:= "DB_Alarms".VibCritical,
	           SafetyOk => "DB_Status".Safety.SafetyOk,
	           PermitMotion => "DB_Status".Safety.PermitMotion,
	           TripActive => "DB_Status".Safety.TripActive, // TripActive znamena "bezpecne odpojeni vykonovych vystupu systemu"
	           TripCode => "DB_Status".Safety.TripCode,
	           StatusText => "DB_Status".Safety.StatusText
	);


	"Spindel"(HMI_Start:= "DB_HMI".Spindle.Start,
	          HMI_Stop:="DB_HMI".Spindle.Stop,
	          HMI_ResetFault:="DB_HMI".Spindle.ResetFault,
	          HMI_Speed_RPM:="DB_HMI".Spindle.Speed_RPM,
	          PermitMotion:="DB_Status".Safety.PermitMotion,
	          EmergencyStop:="DB_IO".DI.EmergencyStop,
	          ExternalFaultIn:="DB_IO".DI.ExternalFault,
	          SpeedMax_RPM:=18000.0,
	          AO_MaxVolt:=10.0,
	          RampUp_RPM_per_s:=6000.0,
	          RampDown_RPM_per_s:=9000.0,
	          ResetPulse:=T#300MS,
	          RequireSpeedToRun:=FALSE,
	          DO_RunForward=>"DB_IO".DQ.RunForwardCmd,
	          DO_FaultReset=>"DB_IO".DQ.FaultResetCmd,
	          DO_MultiSpeed1=>"DB_IO".DQ.MultiSpeed1,
	          DO_ExternalFault=>"DB_IO".DQ.ExternalFault,
	          AQ1_Voltage_0_10V=>"DB_IO".AQ.SpeedVoltage,
	          RunLatched=>"DB_Status".Spindel.RunLatched,
	          TripActive=>"DB_Status".Spindel.TripActive,
	          State=>"DB_Status".Spindel.State,
	          StatusText=>"DB_Status".Spindel.StatusText);

	//******************************************************************
	// AUTO-RESET Spindle pulse bits (v OB1, hned po volání Spindel FB)
	//******************************************************************
	IF "DB_HMI".Spindle.Start THEN
		"DB_HMI".Spindle.Start := FALSE;
	END_IF;
	IF "DB_HMI".Spindle.Stop THEN
		"DB_HMI".Spindle.Stop := FALSE;
	END_IF;

	//******************************************************************
	// LATCH Start/Stop requestu z HMI do runtime DB (OB1 je rychly)
	// Chrani hrany StartTest/StopTest pred ztratou pri OB30=1000ms.
	//******************************************************************
	IF "DB_LogConfig".StartTest THEN
		"DB_LogRuntime".StartReqLatched := TRUE;
	END_IF;
	IF "DB_LogConfig".StopTest THEN
		"DB_LogRuntime".StopReqLatched := TRUE;
		"DB_LogRuntime".StopSequenceActive := TRUE;
	END_IF;

	//******************************************************************
	// CALL OTHER FB BLOCKS
	//******************************************************************
	"FB_SafetyButtons_DB"(DI0_AuxSafetyRelay:="DB_IO".DI.SafetyRelayAuxOk,
	                      DI1_SafetyButton:="DB_IO".DI.EmergencyStop,
	                      DQ0_LED=>"DB_IO".DQ.ResetButtonLed,
	                      DQ1_LED=>"DB_IO".DQ.EmergencyStopButtonLed);

	// ----------------------------------------------------------------
	// FAZE 2: Davkovy zapis logu na SD kartu
	// FlushPending nebo FinalFlush spusti stavovy automat LogFlushToSd.
	// ----------------------------------------------------------------
	// FAZE 2: Davkovy zapis logu na SD kartu
	// FlushPending nebo FinalFlush spusti stavovy automat LogFlushToSd.
	// Po dokonceni AckFlush resetuje FlushPending ve FB_LogManager.
	// ----------------------------------------------------------------
	"LogFlushToSd"(
		Enable          := "DB_LogConfig".Enable,
		FlushRequest    := "LogManager".FlushPending,
		FinalFlush      := NOT "DB_LogRuntime".TestActive AND "LogManager".FlushPending,
		MaxRowsPerFlush := 50,
		RetryLimit      := 3
	);

	//******************************************************************
	// AUTO START LabPSU - deterministicky pri nabehu TestActive (ne jen edge)
	//******************************************************************
	IF "DB_LogRuntime".TestActive AND NOT "DB_LogRuntime".TestActivePrev THEN
		"DB_HMI".LabPSU.Enable := TRUE;
		"DB_HMI".LabPSU.Mode := 2;  // SINE_DEBUG
		"DB_LogRuntime".LastStopLogSaved := FALSE;
	END_IF;

	//******************************************************************
	// STOP COMPLETE - po final flush nastav defaulty pro dalsi test
	//******************************************************************
	IF "DB_LogRuntime".StopSequenceActive
		AND NOT "DB_LogRuntime".TestActive
		AND NOT "LogManager".FlushPending
		AND NOT "LogFlushToSd".AckFlush THEN
		"DB_HMI".LabPSU.Enable := FALSE;
		"DB_HMI".LabPSU.Mode := 2;  // dalsi AUTO startuje v SINE rezimu
		"DB_HMI".Spindle.Speed_RPM := 0.0;
		"DB_LogRuntime".Elapsed_s := 0.0;
		"DB_LogRuntime".ElapsedTime_HMI := '000:00:00';
		"DB_LogRuntime".TimeDisplay_HMI := CONCAT(
			IN1 := "DB_LogRuntime".ElapsedTime_HMI,
			IN2 := CONCAT(IN1 := ' / ', IN2 := "DB_LogRuntime".TargetTime_HMI)
		);
		"DB_LogRuntime".LastStopLogSaved := "DB_LogRuntime".LastFlushOk;
		"DB_LogRuntime".StopSequenceActive := FALSE;
	END_IF;

	//******************************************************************
	// AUTO STOP - Test timeout handling - VYPNUTO (test bezi do nekonecna)
	// Kdyz test dosahl casu TestDuration_s, automaticky zastav vse
	//******************************************************************
	// IF "LogManager".TestTimeoutReached THEN
	// 	// Automaticky zastav vreteno - puls se vygeneruje pres HMI bit
	// 	// (FB_DriveCtrl ma edge detection, takze staci nastavit a zresetovat v dalsim cyklu)
	// 	IF NOT "DB_HMI".Spindle.Stop THEN
	// 		"DB_HMI".Spindle.Stop := TRUE;
	// 	ELSE
	// 		"DB_HMI".Spindle.Stop := FALSE;
	// 		"LogManager".TestTimeoutReached := FALSE;  // Reset timeout flag
	// 	END_IF;
	//
	// 	// Vypni laboratorni zdroj
	// 	"DB_HMI".LabPSU.Enable := FALSE;
	//
	// 	// Stop log (puls) - FlushPending uz je TRUE z FB_LogManager
	// 	// TestActive uz je FALSE z FB_LogManager
	// END_IF;

	//******************************************************************
	// HMI HELPER - Status panel color (Basic Panel limitation)
	// Priority: RED (trip) > AMBER (warning) > BLUE (running) > GREEN (ready)
	//******************************************************************
	//******************************************************************
	IF "DB_Status".Safety.TripActive THEN
		"DB_Status".HMI_StatusColor := 2;  // RED - error/trip active
		"DB_Status".HMI_StatusText := 'ERROR - TRIP ACTIVE';
	ELSE
		IF "DB_LogRuntime".TestActive THEN
			IF "DB_HMI".Spindle.Speed_RPM <= 0.0 THEN
				"DB_Status".HMI_StatusColor := 3;  // AMBER - running but setpoint is zero
				"DB_Status".HMI_StatusText := 'RUNNING - RPM=0';
			ELSE
				"DB_Status".HMI_StatusColor := 1;  // GREEN - test running
				"DB_Status".HMI_StatusText := 'TEST RUNNING';
			END_IF;
		ELSE
			"DB_Status".HMI_StatusColor := 0;  // GREEN - ready/stopped
			IF "DB_LogRuntime".LastStopLogSaved THEN
				"DB_Status".HMI_StatusText := 'READY - LOG SAVED';
			ELSE
				"DB_Status".HMI_StatusText := 'TEST READY';
			END_IF;
		END_IF;
	END_IF;

	"DB_LogRuntime".TestActivePrev := "DB_LogRuntime".TestActive;

	//******************************************************************
	// CONVERT IO - AŽ na konci, po všech FB!
	//******************************************************************
	"FC_ConvertIO"();

	//******************************************************************
	// IO MAP WRITE - zapisat vypocitane vystupy na fyzicke vystupy
	//******************************************************************
	"FC_IO_Map_Write"();
END_ORGANIZATION_BLOCK

